{attribute addProperty BoxType "EKM1101-0000-0016"}
{attribute addProperty Id "AdsAddrAT %I*AMSADDR6480DcOutputShiftAT %I*DINT3240DcInputShiftAT %I*DINT3240StateAT %I*UINT1620"}
{attribute addProperty CRC "199153599"}
{attribute addProperty SizeInBites "144"}
{attribute addProperty SizeInBytes "18"}
TYPE InfoData_0BDED7BF :
STRUCT
	{attribute addProperty Name "AdsAddr"}
	AdsAddr AT %I* : AMSADDR;
	{attribute addProperty Name "DcOutputShift"}
	DcOutputShift AT %I* : DINT;
	{attribute addProperty Name "DcInputShift"}
	DcInputShift AT %I* : DINT;
	{attribute addProperty Name "State"}
	State AT %I* : UINT;
END_STRUCT
END_TYPE

(* stored: Version 1.2.0.0, ProductVersion 3.1.4024.9
   DUT InfoData_0BDED7BF: Id {c0def2d2-6afa-4037-bd85-5e2c3dc75ca6} *)
